FUNCTION_BLOCK GenerateTimeData_TEST EXTENDS TcUnit.FB_TestSuite
VAR_INPUT
END_VAR
VAR_OUTPUT
END_VAR
VAR
END_VAR

CheckStringFormat();

METHOD CheckStringFormat
VAR_INPUT
END_VAR
VAR_INST
	sut		:	GenerateTimeData;
	expected:	STRING;
	result 	: 	STRING;
END_VAR
sut();

TEST('CheckStringFormat');

expected := CONCAT('-', TO_STRING(sut.timeAsSystemTime.wYear));
IF sut.timeAsSystemTime.wMonth < 10 THEN expected := CONCAT(expected, '0'); END_IF
expected := CONCAT(expected, TO_STRING(sut.timeAsSystemTime.wMonth));
IF sut.timeAsSystemTime.wDay < 10 THEN expected := CONCAT(expected, '0'); END_IF
expected := CONCAT(expected, TO_STRING(sut.timeAsSystemTime.wDay));
expected := CONCAT(expected, '-');
IF sut.timeAsSystemTime.wHour < 10 THEN expected := CONCAT(expected, '0'); END_IF
expected := CONCAT(expected, TO_STRING(sut.timeAsSystemTime.wHour));
expected := CONCAT(expected, ':');
IF sut.timeAsSystemTime.wMinute < 10 THEN expected := CONCAT(expected, '0'); END_IF
expected := CONCAT(expected, TO_STRING(sut.timeAsSystemTime.wMinute));
expected := CONCAT(expected, ':');
IF sut.timeAsSystemTime.wSecond < 10 THEN expected := CONCAT(expected, '0'); END_IF
expected := CONCAT(expected, TO_STRING(sut.timeAsSystemTime.wSecond));
expected := CONCAT(expected, '-');

result := sut.ToString('-YYYYMMDD-hh:mm:ss-');
	
IF sut.Done THEN
	AssertEquals(
		Expected 	:= 	expected,
		Actual 		:=  result,
		Message		:=	'Time formatting failed.'
	);

	TEST_FINISHED();
END_IF
END_METHOD

END_FUNCTION_BLOCK

(* stored: Version 1.1.0.1
   POU GenerateTimeData_TEST: Id {7d8824eb-9fb9-4da8-9874-6ae610f7d88c}, SpecialFunc None
   Method CheckStringFormat: Id {5a0ae825-ada9-4cee-957b-1cdb64d42545} *)
